FUNCTION F_CompareObjects : BOOL
VAR_INPUT
    ipObject1:      I_Object;
    ipObject2:      I_Object;
END_VAR
VAR
END_VAR

IF ipObject1 = ipObject2 THEN
    F_CompareObjects := TRUE;
END_IF

END_FUNCTION

(* stored: Version 1.1.0.1, ProductVersion 3.1.4024.12
   POU F_CompareObjects: Id {fc180723-9f9e-440c-aaf8-4cd3ca30bb42}, SpecialFunc None *)
